SUBAPPLICATION Uebung_011e_PHYSA (* Numeric Value Input I1 Durchschleifen auf N3 (Software Scale via NumericObjectPool_S) *)
  (* Standard: 61499-2; Description: Copyright (c) 2023 Meisterschulen am Ostbahnhof This program and the accompanying materials are made available under the terms of the Eclipse Public License 2.0 which is available at https://www.eclipse.org/legal/epl-2.0/ SPDX-License-Identifier: EPL-2.0 *)
  (* Version 1.0, 2026-04-14, Franz Höpfinger, Meisterschulen am Ostbahnhof, initial API and implementation and/or initial documentation *)
  PACKAGE Uebungen;
  IMPORT Uebungen::const::UT::DefaultPool::InputNumber_I1;
  IMPORT Uebungen::const::UT::DefaultPool_Numeric::OutputNumber_N3;
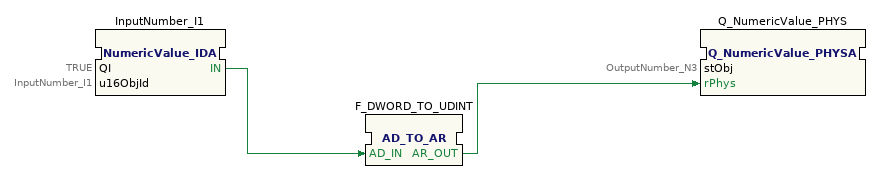
  (* Beispiel: I1-Eingabe 10 → F_RAW_TO_PHYS(I1) → 10.0 → Q_NumericValue_PHYS(N3) → N3 zeigt 10.00. die beiden Namespaces sind INKOMPATIBEL !!! *)
  (* Uebungen::const::UT::DefaultPool_Numeric::OutputNumber_N3 *)
  (* Uebungen::const::UT::DefaultPool::InputNumber_I1 *)
  FBS
    InputNumber_I1 : isobus::UT::io::NumericValue::NumericValue_IDA(QI := TRUE, u16ObjId := InputNumber_I1);
    F_DWORD_TO_UDINT : adapter::conversion::unidirectional::AD_TO_AR;
    Q_NumericValue_PHYS : isobus::UT::Q::Q_NumericValue_PHYSA(stObj := OutputNumber_N3);
  END_FBS
  ADAPTER_CONNECTIONS
    F_DWORD_TO_UDINT.AR_OUT TO Q_NumericValue_PHYS.rPhys;
    InputNumber_I1.IN TO F_DWORD_TO_UDINT.AD_IN;
  END_CONNECTIONS
END_SUBAPPLICATION
